TYPE TcoOmnicore_Inputs_v_1_x_x :
STRUCT
	Inputs AT %I* : ARRAY[0..63] OF BYTE;
END_STRUCT
END_TYPE

(* stored: Version 1.1.0.1, ProductVersion 3.1.4024.12
   DUT TcoOmnicore_Inputs_v_1_x_x: Id {836289e2-aa24-036a-3f09-664edf124071} *)
